FUNCTION_BLOCK FB_Mediator IMPLEMENTS I_Module

VAR
	aPeersConnected : ARRAY[1..nMAX_PEER_NUMBER] OF ST_PeerAccount;
	aLogMessages :  ARRAY[1..nMAX_LOG_MESSAGES] OF T_MaxString;
	aPeerUnits : ARRAY[1..nMAX_PEER_NUMBER] OF ST_LinkedListUnit;
	aLogUnits : ARRAY[1..nMAX_LOG_MESSAGES] OF ST_LinkedListUnit;
	
	fbPeersList : FB_PeerLinkedList;
	//fbLogList : FB_Logging;
	
	nStackPointer : UINT := 1;
	bAtLeastOnePeerConnected : BOOL;
	bInit : BOOL;
	i : UINT;
	
	stTestUnit : ST_LinkedListUnit;
	pTestMessage : POINTER TO ST_Message;
	stEmptyMessage : ST_MESSAGE;
	sModuleName : STRING;
	
	//DEBUG:
	//If one of the following variables becomes TRUE, investigation of the cause is mandatory
//--------------------------------------------------------------------------------------------
	bFailedToRelocateToTail : BOOL;
	bNullExceptionWhileDispatching : BOOL;
	bNullExceptionWhileCheckingMailbox : BOOL;
//--------------------------------------------------------------------------------------------


END_VAR
VAR CONSTANT
	
END_VAR

M_Init();
M_CheckMailboxes();
M_DispatchMessages();


PROPERTY AccessModuleName : STRING
GET
AccessModuleName := sModuleName;
END_GET
SET
sModuleName := AccessModuleName;
END_SET
END_PROPERTY

METHOD PUBLIC M_AddPeer : E_MediatorReturnCode
VAR_INPUT
	in_iPeer : I_Peer;
END_VAR
VAR
	i : UINT;
	
END_VAR
IF NOT fbPeersList.bInit THEN
	RETURN;
END_IF

IF nStackPointer > nMAX_PEER_NUMBER THEN
	M_AddPeer := E_MediatorReturnCode.eMAX_NUMBER_OF_CONNECTED_PEERS;
	RETURN;
END_IF

FOR i := 1 TO nMAX_PEER_NUMBER DO
	IF aPeersConnected[i].iPeer = in_iPeer THEN
		M_AddPeer := E_MediatorReturnCode.ePEER_ALREADY_CONNECTED;
		RETURN;	
	END_IF
END_FOR

aPeersConnected[nStackPointer].iPeer := in_iPeer;
aPeersConnected[nStackPointer].rMailbox Ref= in_iPeer.M_RetrieveMailbox();

fbPeersList.M_AddPeerToTail
(
	pPeerToAdd := ADR(aPeersConnected[nStackPointer]),
	pUnitToAdd := ADR(aPeerUnits[nStackPointer])
);

nStackPointer := nStackPointer + 1;

bAtLeastOnePeerConnected := TRUE;

M_AddPeer := E_MediatorReturnCode.ePEER_CONNECTED;
END_METHOD

METHOD PRIVATE M_CheckMailboxes : BOOL

VAR
	nSendersAccount : UINT;
	nSendersStackPointer : UINT;
	stMessageToAdd : ST_Message;
	pPeer : POINTER TO ST_PeerAccount;
END_VAR
IF NOT bAtLeastOnePeerConnected THEN
	RETURN;
END_IF 

FOR nSendersAccount := 1 TO nStackPointer-1 DO
	
(*
	IF nSendersAccount = 1 THEN
		fbPeersList.pGetCurrent := fbPeersList.pHead;
		fbPeersList.nGetNextPosition := 1;
	END_IF
*)

	pPeer :=  fbPeersList.M_GetNextPeer();
	
	IF pPeer = NULL THEN
		//Report null exception
		bNullExceptionWhileCheckingMailbox := TRUE;
		CONTINUE;
	END_IF
	
	IF pPeer^.rMailbox.bMessageSent THEN
		pPeer^.rMailbox.bMessageSent := FALSE;
	END_IF;
	
	//If sender has a message in its outbox, add the message to the list of messages
	//The oldest message always in front of the list (FIFO)
	IF pPeer^.rMailbox.bSendingMessage THEN
		
		nSendersStackPointer := pPeer^.nStackPointer;
		// If the senders account has less then X messages, add the outgoing message to the message list 
		IF nSendersStackPointer <= nMAX_DATA_ELEMENTS THEN
	
			stMessageToAdd := pPeer^.rMailbox.stOutbox;
			
			pPeer^.bMailboxFull := FALSE;
			pPeer^.aMessages[nSendersStackPointer] := stMessageToAdd;		
			pPeer^.nStackPointer := nSendersStackPointer + 1;		
			pPeer^.bMailboxEmpty := FALSE;		
			pPeer^.rMailbox.bSendingMessage := FALSE;
			pPeer^.rMailbox.stOutbox := stEmptyMessage;
	
			//Will be true for only one cycle
			pPeer^.rMailbox.bMessageSent := TRUE;
			
		ELSE
			
			//Mailbox contains more than X messages
			pPeer^.bMailboxFull := TRUE;
			
		END_IF
		
	END_IF
	
END_FOR
END_METHOD

METHOD PRIVATE M_DeleteMessageFromSendersAccount : BOOL
VAR_INPUT
	in_pSenderPeer : POINTER TO ST_PeerAccount;
END_VAR
VAR
	stEmptyMessage : ST_MESSAGE;
	nSendersStackPointer : UINT;
	i : UINT;
END_VAR
IF in_pSenderPeer^.bMailboxEmpty THEN
	RETURN;
END_IF 

nSendersStackPointer := in_pSenderPeer^.nStackPointer;
in_pSenderPeer^.nStackPointer := nSendersStackPointer - 1;

//Only one message was in the list
IF in_pSenderPeer^.nStackPointer = 1 THEN
	
	//Remove oldest message from list
	in_pSenderPeer^.aMessages[1] := stEmptyMessage;
	in_pSenderPeer^.bMailboxEmpty := TRUE;
ELSE
	//Move all the messages by one 
	FOR i := 2 TO nSendersStackPointer-1 DO 
		in_pSenderPeer^.aMessages[i - 1] := 
			in_pSenderPeer^.aMessages[i];
	END_FOR
	
	//Remove newest message from list
	in_pSenderPeer^.aMessages[nSendersStackPointer-1] := stEmptyMessage;
	
END_IF
END_METHOD

METHOD PRIVATE M_DispatchMessages 
VAR_INPUT
END_VAR
VAR_OUTPUT
	
END_VAR
VAR
	nSenderPeer : UINT;
	nReceiverPeer : UINT;
	
	pPeer : POINTER TO ST_PeerAccount;
	pUnit : POINTER TO ST_LinkedListUnit;
	
	nPeerListPosition : UINT;
END_VAR

VAR_INST

END_VAR
IF 	NOT bAtLeastOnePeerConnected 
	OR fbPeersList.M_GetCurrentPosition() = 0
	THEN
	
	RETURN;
END_IF 

FOR nSenderPeer := 1 TO nStackPointer-1 DO
(*	
	IF nSenderPeer = 1 THEN
		fbPeersList.pGetCurrent := fbPeersList.pHead;
		fbPeersList.nGetNextPosition := 1;
	END_IF
*)
	pPeer :=  fbPeersList.M_GetNextPeer();
	
	IF pPeer = NULL THEN
		//Report null exception
		bNullExceptionWhileDispatching := TRUE;
		CONTINUE;
	END_IF
	
	//Check if peer has mail to send
	IF NOT pPeer^.bMailboxEmpty THEN
		
		//Result 0 means peer not found
		nReceiverPeer := M_FindPeer( M_GetReceiverPeerId( pPeer ) );
		
		IF nReceiverPeer > 0 THEN
			
			//Sends the message only when the receiver has emptied its own mailbox
			IF 	NOT aPeersConnected[nReceiverPeer].rMailbox.bNewMessageAvail
				THEN				
				
				M_SendMessage
				(
					in_nReceiverPeer := nReceiverPeer,
					in_pSenderPeer := pPeer 
				);
				
				IF pPeer^.aMessages[1].eDeliveryStatus = E_DeliveryStatus.eDELIVERY_REJECTED THEN
					
					fbLogList.M_Info(
						in_iModule:=THIS^,
						in_sMessage:= 
							F_Concat8(
								'Peer ', 
								GTL.gtlPeers[ pPeer^.iPeer.M_GetPeerId() ],
								' sending message back to Peer ',
								GTL.gtlPeers[ M_GetReceiverPeerId( pPeer ) ],
								': ',
								GTL.gtlMessages[ pPeer^.aMessages[1].eMessage ],
								';Delivery status: ',
								GTL.gtlDeliveryStatus[ pPeer^.aMessages[1].eDeliveryStatus ]						
							) 	
					);
					
				ELSE
					
					fbLogList.M_Info(
						in_iModule:=THIS^,
						in_sMessage:= 
							F_Concat8(
								'Peer ', 
								GTL.gtlPeers[ pPeer^.iPeer.M_GetPeerId() ],
								' sending following message to Peer ',
								GTL.gtlPeers[ M_GetReceiverPeerId( pPeer ) ],
								': ',
								GTL.gtlMessages[ pPeer^.aMessages[1].eMessage ],
								';Delivery status: ',
								GTL.gtlDeliveryStatus[ E_DeliveryStatus.eDELIVERY_OK ]						
							) 	
					);
					
				END_IF

				
				M_DeleteMessageFromSendersAccount(in_pSenderPeer := pPeer);	
							
				pPeer^.eDispatchRoutineReturnCode := eMESSAGE_DISPATCHED;
				
				bFailedToRelocateToTail S= NOT fbPeersList.M_RelocateToTail();


			ELSE
				
				pPeer^.eDispatchRoutineReturnCode := eMESSAGE_NOT_DISPATCHED;
				pPeer^.aMessages[1].eDeliveryStatus := E_DeliveryStatus.eRECEIVERS_MAILBOX_NOT_EMPTY;
				
				fbLogList.M_Info(
					in_iModule:=THIS^,
					in_sMessage:= 
						F_Concat8(
							'Peer ', 
							GTL.gtlPeers[ pPeer^.iPeer.M_GetPeerId() ],
							' failed to send following message to Peer ',
							GTL.gtlPeers[ M_GetReceiverPeerId( pPeer ) ],
							': ',
							GTL.gtlMessages[ pPeer^.aMessages[1].eMessage ],
							';Delivery status: ',
							GTL.gtlDeliveryStatus[ pPeer^.aMessages[1].eDeliveryStatus ]						
						) 	
				);	
				
			END_IF
			
		ELSE
			
			// Report peer not found;	
			
			fbLogList.M_Info(
				in_iModule:=THIS^,
				in_sMessage:= 
					F_Concat8(
						'Peer ', 
						GTL.gtlPeers[ pPeer^.iPeer.M_GetPeerId() ],
						' failed to send following message to Peer ',
						GTL.gtlPeers[ M_GetReceiverPeerId( pPeer ) ],
						': ',
						GTL.gtlMessages[ pPeer^.aMessages[1].eMessage ],
						';Delivery status: ',
						GTL.gtlDeliveryStatus[ E_DeliveryStatus.ePEER_NOT_FOUND ]						
					) 	
			);
			M_DeleteMessageFromSendersAccount(in_pSenderPeer := pPeer);	
			pPeer^.eDispatchRoutineReturnCode := ePEER_NOT_FOUND;
			
		END_IF
				
	END_IF
	
END_FOR
END_METHOD

METHOD PRIVATE M_FindPeer : UINT
VAR_INPUT
	in_ePeer : E_PeersList;
END_VAR
VAR
	i : UINT;
END_VAR
IF 	NOT bAtLeastOnePeerConnected 
	OR in_ePeer = NULL 
	THEN
	
	RETURN;
	
END_IF 

//Check if receiver peer is in the peers list and return position of peer in the list
FOR i := 1 TO nStackPointer - 1 DO
	
	IF aPeersConnected[i].iPeer.M_GetPeerId() = in_ePeer THEN
		
		M_FindPeer := i;
		RETURN;
		
	END_IF
	
END_FOR

M_FindPeer := 0;
END_METHOD

METHOD PRIVATE M_GetReceiverPeerId : E_PeersList
VAR_INPUT
	in_pSenderPeer : POINTER TO ST_PeerAccount;
END_VAR
VAR
	pMessage : POINTER TO ST_Message;
END_VAR
//Extract receivers Id from the oldest message in the list
M_GetReceiverPeerId := in_pSenderPeer^.aMessages[1].eToPeer;
END_METHOD

METHOD PRIVATE M_Init : BOOL
VAR_INPUT
END_VAR
fbPeersList.M_InitLinkedList(aPeerUnits);
fbLogList.M_InitLinkedList(aLogUnits);
fbLogList(in_sPath := GVL_SystemParams.sLogPath);

IF NOT bInit THEN
	bInit := TRUE;
	
	fbLogList.AccessLoggingSeverity := eALL;
	
	FOR i := 1 TO nMAX_LOG_MESSAGES DO
		aLogUnits[i].pVoid := ADR(aLogMessages[i]);
		fbLogList.M_AddToTail(ADR(aLogUnits[i]));
	END_FOR

END_IF
END_METHOD

METHOD PUBLIC M_IsPeerConnected : BOOL
VAR_INPUT
	in_ePeer : E_PeersList;
END_VAR
VAR
	i : UINT;
END_VAR
FOR i := 1 TO nMAX_PEER_NUMBER DO
	
	IF aPeersConnected[i].iPeer.M_GetPeerId() = in_ePeer THEN
		
		M_IsPeerConnected := TRUE;
		RETURN;
		
	END_IF
	
END_FOR
END_METHOD

METHOD PRIVATE M_SendMessage : BOOL
VAR_INPUT
	in_nReceiverPeer : UINT;
	in_pSenderPeer : POINTER TO ST_PeerAccount;
END_VAR
//Dispatch mail after the FIFO principle
aPeersConnected[in_nReceiverPeer].rMailbox.stInbox := in_pSenderPeer^.aMessages[1];
aPeersConnected[in_nReceiverPeer].rMailbox.bNewMessageAvail := TRUE;
END_METHOD

END_FUNCTION_BLOCK

(* stored: Version 1.1.0.1, ProductVersion 3.1.4022.16
   POU FB_Mediator: Id {c5574a95-b005-4b8b-ba18-453adb328f12}, SpecialFunc None
   Property AccessModuleName: Id {1c5546e5-c0d1-446f-9ee3-8a3984b7900d}
   Get Get: Id {e5072c3c-8814-450b-a9db-439e17ad00d1}
   Set Set: Id {54e52490-0b5f-4f93-ba3a-29419aa39937}
   Method M_AddPeer: Id {694e1e7b-7df5-4562-92ab-e389ee720bcc}
   Method M_CheckMailboxes: Id {cd0b5dd7-0ae3-4858-8ff7-ce85195c1ca9}
   Method M_DeleteMessageFromSendersAccount: Id {9f20e6c9-acb9-4365-ba5d-c0831e56f4b4}
   Method M_DispatchMessages: Id {8caccc8f-9c76-40c6-b08f-e8828ce973c6}
   Method M_FindPeer: Id {878caac1-d47b-4a31-9e53-2db987497e7a}
   Method M_GetReceiverPeerId: Id {22257351-27a0-43bb-96ee-bf162d2f9dfc}
   Method M_Init: Id {31fbd38e-fc0f-40dc-bfd5-42b45e9fd264}
   Method M_IsPeerConnected: Id {9f12470a-c2b8-4395-87f5-2eeef52e26d8}
   Method M_SendMessage: Id {99be8876-3430-43f6-82fc-8cdde1ca3f33} *)
